FUNCTION_BLOCK BargraphSplitFS (* Visualizes a signed REAL value as two adjacent Linear Bar Graphs (unsigned magnitude fills meeting at a shared zero point) *)
  (* Standard: ISO 11783-6; Description: Copyright (c) 2026 Meisterschulen am Ostbahnhof This program and the accompanying materials are made available under the terms of the Eclipse Public License 2.0 which is available at https://www.eclipse.org/legal/epl-2.0/ SPDX-License-Identifier: EPL-2.0 Wraps two Q_NumericValue_PHYS instances (ISO 11783-6 F.22) that command a pair of adjacent Linear Bar Graph objects (Annex B.11.3), given an arbitrary signed REAL value. stObj is snapshotted once at INIT via F_MOVE, matching the ScrollFS/PositionMarkerFS pattern. rValue > 0 clamps to [0, r32MaxMagnitude] and is written to the right side; the left side receives 0. rValue < 0 is negated (F_MUL by -1.0), clamped the same way, and written to the left side; the right side receives 0. xOverRight/xOverLeft report a magnitude exceeding r32MaxMagnitude on the respective side. There are deliberately no xUnder outputs: falling below r32MinMagnitude (0) on the currently-inactive side is the normal resting state during ordinary operation, not a diagnostic condition. *)
  (* Version 1.0, 2026-09-05, Franz Höpfinger, Meisterschulen am Ostbahnhof, initial API and implementation and/or initial documentation *)
  PACKAGE isobus::UT::Q;
  IMPORT isobus::utils::bargraph::BargraphSplit_S;
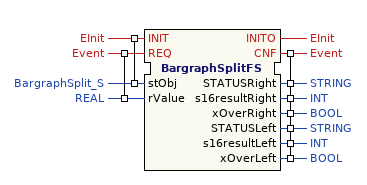
  EVENT_INPUT
    INIT : EInit WITH stObj; (* Service Initialization *)
    REQ WITH rValue; (* Display a new signed value *)
  END_EVENT
  EVENT_OUTPUT
    INITO : EInit; (* Initialization Confirm *)
    CNF WITH STATUSRight, s16resultRight, xOverRight, STATUSLeft, s16resultLeft, xOverLeft; (* Confirmation of Requested Service *)
  END_EVENT
  VAR_INPUT
    stObj : isobus::utils::bargraph::BargraphSplit_S; (* Split-bargraph object pool properties (left/right Bargraph refs, shared magnitude bounds), snapshotted at INIT *)
    rValue : REAL; (* Signed physical value to display - from any source, not limited to NumericValue_PHYS *)
  END_VAR
  VAR_OUTPUT
    STATUSRight : STRING; (* Service Status - passthrough from the internal right-side Q_NumericValue_PHYS *)
    s16resultRight : INT; (* retval - passthrough from the internal right-side Q_NumericValue_PHYS *)
    xOverRight : BOOL; (* rValue exceeded stObj.r32MaxMagnitude and the right side was clamped *)
    STATUSLeft : STRING; (* Service Status - passthrough from the internal left-side Q_NumericValue_PHYS *)
    s16resultLeft : INT; (* retval - passthrough from the internal left-side Q_NumericValue_PHYS *)
    xOverLeft : BOOL; (* -rValue exceeded stObj.r32MaxMagnitude and the left side was clamped *)
  END_VAR
  FBS
    Snap : iec61131::selection::F_MOVE; {SET_ATTRIBUTE(DataType, isobus::utils::bargraph::BargraphSplit_S)}
    ClampRight : logiBUS::signalprocessing::clamp::F_ClampReal;
    NumRight : isobus::UT::Q::Q_NumericValue_PHYS;
    NegateValue : iec61131::arithmetic::F_MUL(IN2 := REAL#-1.0);
    ClampLeft : logiBUS::signalprocessing::clamp::F_ClampReal;
    NumLeft : isobus::UT::Q::Q_NumericValue_PHYS;
  END_FBS
  EVENT_CONNECTIONS
    INIT TO Snap.REQ;
    Snap.CNF TO NumRight.INIT;
    NumRight.INITO TO NumLeft.INIT;
    NumLeft.INITO TO INITO;
    REQ TO ClampRight.REQ;
    ClampRight.CNF TO NumRight.REQ;
    NumRight.CNF TO NegateValue.REQ;
    NegateValue.CNF TO ClampLeft.REQ;
    ClampLeft.CNF TO NumLeft.REQ;
    NumLeft.CNF TO CNF;
  END_CONNECTIONS
  DATA_CONNECTIONS
    stObj TO Snap.IN;
    Snap.OUT.stRight TO NumRight.stObj;
    Snap.OUT.stLeft TO NumLeft.stObj;
    rValue TO ClampRight.rIn;
    Snap.OUT.r32MinMagnitude TO ClampRight.rMin;
    Snap.OUT.r32MaxMagnitude TO ClampRight.rMax;
    ClampRight. TO NumRight.rPhys;
    rValue TO NegateValue.IN1;
    NegateValue.OUT TO ClampLeft.rIn;
    Snap.OUT.r32MinMagnitude TO ClampLeft.rMin;
    Snap.OUT.r32MaxMagnitude TO ClampLeft.rMax;
    ClampLeft. TO NumLeft.rPhys;
    NumRight.STATUS TO STATUSRight;
    NumRight.s16result TO s16resultRight;
    ClampRight.xOver TO xOverRight;
    NumLeft.STATUS TO STATUSLeft;
    NumLeft.s16result TO s16resultLeft;
    ClampLeft.xOver TO xOverLeft;
  END_CONNECTIONS
END_FUNCTION_BLOCK
